// TIA Portal V21 export
ORGANIZATION_BLOCK "Main"   // OB1, LAD, ProgramCycle
TITLE = "Main Program Sweep (Cycle)"
{ S7_Optimized_Access := 'TRUE' }
// stored: SetENOAutomatically false
   VAR_INPUT
      Initial_Call : Bool;   // Initial call of this OB
      Remanence : Bool;   // =True, if remanent data are available
   END_VAR
   VAR_TEMP
      "EQUIPMENT ID" : Variant;
      "EQUIPMENT ID_1" : Variant;
   END_VAR
   VAR_TEMP   // added for the SCL form of the ladder/FBD networks
      _w1 : Bool;
      _w2 : Bool;
      _w3 : Bool;
      _w4 : Bool;
      _w5 : Bool;
      _w6 : Bool;
      _w7 : Bool;
   END_VAR
BEGIN

REGION Network 1: BLOCK CALL
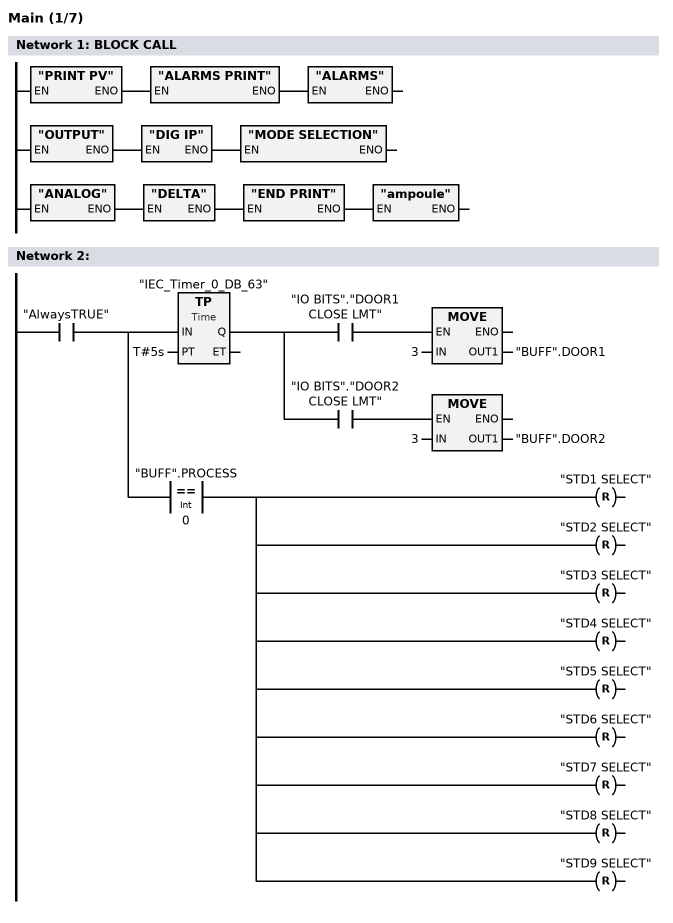
   RUNG wire#powerrail
      "PRINT PV"()
      "ALARMS PRINT"()
      "ALARMS"()
   END_RUNG
   RUNG wire#powerrail
      "OUTPUT"()
      "DIG IP"()
      "MODE SELECTION"()
   END_RUNG
   RUNG wire#powerrail
      "ANALOG"()
      "DELTA"()
      "END PRINT"()
      "ampoule"()
   END_RUNG
   // the same network as SCL:
   "PRINT PV"(ENO => #_w1);
   "ALARMS PRINT"(EN := #_w1, ENO => #_w2);
   IF #_w2 THEN "ALARMS"(); END_IF;
   "OUTPUT"(ENO => #_w3);
   "DIG IP"(EN := #_w3, ENO => #_w4);
   IF #_w4 THEN "MODE SELECTION"(); END_IF;
   "ANALOG"(ENO => #_w5);
   "DELTA"(EN := #_w5, ENO => #_w6);
   "END PRINT"(EN := #_w6, ENO => #_w7);
   IF #_w7 THEN "ampoule"(); END_IF;
END_REGION

REGION Network 2
   RUNG wire#powerrail
      Contact( "AlwaysTRUE" )
      wire#w1
      { S7_Templates := "time_type := Time" } "IEC_Timer_0_DB_63".TP(pt := T#5s, et =>)
      wire#w2
      Contact( "IO BITS"."DOOR1 CLOSE LMT" )
      Move(in := 3, out1 => "BUFF".DOOR1)
   END_RUNG
   RUNG wire#w2
      Contact( "IO BITS"."DOOR2 CLOSE LMT" )
      Move(in := 3, out1 => "BUFF".DOOR2)
   END_RUNG
   RUNG wire#w1
      { S7_Templates := "SrcType := Int" } EQ_Contact(in1 := "BUFF".PROCESS, in2 := 0)
      wire#w3
      R_Coil( "STD1 SELECT" )
   END_RUNG
   RUNG wire#w3
      R_Coil( "STD2 SELECT" )
   END_RUNG
   RUNG wire#w3
      R_Coil( "STD3 SELECT" )
   END_RUNG
   RUNG wire#w3
      R_Coil( "STD4 SELECT" )
   END_RUNG
   RUNG wire#w3
      R_Coil( "STD5 SELECT" )
   END_RUNG
   RUNG wire#w3
      R_Coil( "STD6 SELECT" )
   END_RUNG
   RUNG wire#w3
      R_Coil( "STD7 SELECT" )
   END_RUNG
   RUNG wire#w3
      R_Coil( "STD8 SELECT" )
   END_RUNG
   RUNG wire#w3
      R_Coil( "STD9 SELECT" )
   END_RUNG
   // the same network as SCL:
   "IEC_Timer_0_DB_63".TP(IN := "AlwaysTRUE", PT := T#5s);
   IF "IEC_Timer_0_DB_63".Q AND "IO BITS"."DOOR1 CLOSE LMT" THEN "BUFF".DOOR1 := 3; END_IF;
   IF "IEC_Timer_0_DB_63".Q AND "IO BITS"."DOOR2 CLOSE LMT" THEN "BUFF".DOOR2 := 3; END_IF;
   IF "AlwaysTRUE" AND ("BUFF".PROCESS = 0) THEN
       "STD1 SELECT" := FALSE;
       "STD2 SELECT" := FALSE;
       "STD3 SELECT" := FALSE;
       "STD4 SELECT" := FALSE;
       "STD5 SELECT" := FALSE;
       "STD6 SELECT" := FALSE;
       "STD7 SELECT" := FALSE;
       "STD8 SELECT" := FALSE;
       "STD9 SELECT" := FALSE;
   END_IF;
END_REGION

REGION Network 3: STANDARD1
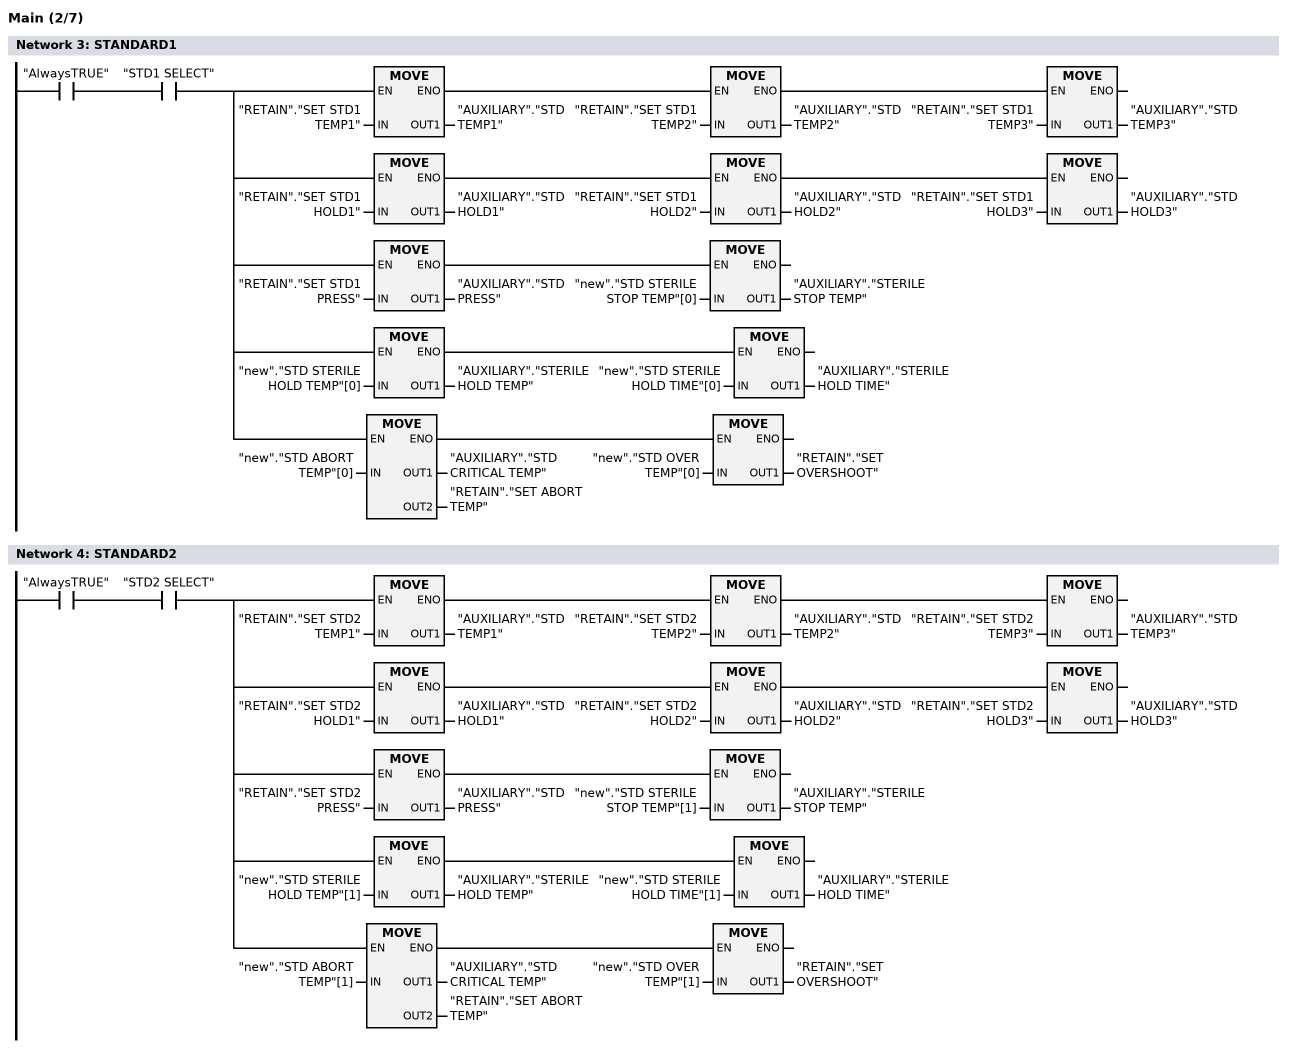
   RUNG wire#powerrail
      Contact( "AlwaysTRUE" )
      Contact( "STD1 SELECT" )
      wire#w1
      Move(in := "RETAIN"."SET STD1 TEMP1", out1 => "AUXILIARY"."STD TEMP1")
      Move(in := "RETAIN"."SET STD1 TEMP2", out1 => "AUXILIARY"."STD TEMP2")
      Move(in := "RETAIN"."SET STD1 TEMP3", out1 => "AUXILIARY"."STD TEMP3")
   END_RUNG
   RUNG wire#w1
      Move(in := "RETAIN"."SET STD1 HOLD1", out1 => "AUXILIARY"."STD HOLD1")
      Move(in := "RETAIN"."SET STD1 HOLD2", out1 => "AUXILIARY"."STD HOLD2")
      Move(in := "RETAIN"."SET STD1 HOLD3", out1 => "AUXILIARY"."STD HOLD3")
   END_RUNG
   RUNG wire#w1
      Move(in := "RETAIN"."SET STD1 PRESS", out1 => "AUXILIARY"."STD PRESS")
      Move(in := "new"."STD STERILE STOP TEMP"[0], out1 => "AUXILIARY"."STERILE STOP TEMP")
   END_RUNG
   RUNG wire#w1
      Move(in := "new"."STD STERILE HOLD TEMP"[0], out1 => "AUXILIARY"."STERILE HOLD TEMP")
      Move(in := "new"."STD STERILE HOLD TIME"[0], out1 => "AUXILIARY"."STERILE HOLD TIME")
   END_RUNG
   RUNG wire#w1
      Move(in := "new"."STD ABORT TEMP"[0], out1 => "AUXILIARY"."STD CRITICAL TEMP", out2 => "RETAIN"."SET ABORT TEMP")
      Move(in := "new"."STD OVER TEMP"[0], out1 => "RETAIN"."SET OVERSHOOT")
   END_RUNG
   // the same network as SCL:
   IF "AlwaysTRUE" AND "STD1 SELECT" THEN
       "AUXILIARY"."STD TEMP1" := "RETAIN"."SET STD1 TEMP1";
       "AUXILIARY"."STD TEMP2" := "RETAIN"."SET STD1 TEMP2";
       "AUXILIARY"."STD TEMP3" := "RETAIN"."SET STD1 TEMP3";
       "AUXILIARY"."STD HOLD1" := "RETAIN"."SET STD1 HOLD1";
       "AUXILIARY"."STD HOLD2" := "RETAIN"."SET STD1 HOLD2";
       "AUXILIARY"."STD HOLD3" := "RETAIN"."SET STD1 HOLD3";
       "AUXILIARY"."STD PRESS" := "RETAIN"."SET STD1 PRESS";
       "AUXILIARY"."STERILE STOP TEMP" := "new"."STD STERILE STOP TEMP"[0];
       "AUXILIARY"."STERILE HOLD TEMP" := "new"."STD STERILE HOLD TEMP"[0];
       "AUXILIARY"."STERILE HOLD TIME" := "new"."STD STERILE HOLD TIME"[0];
       "AUXILIARY"."STD CRITICAL TEMP" := "new"."STD ABORT TEMP"[0];
       "RETAIN"."SET ABORT TEMP" := "new"."STD ABORT TEMP"[0];
       "RETAIN"."SET OVERSHOOT" := "new"."STD OVER TEMP"[0];
   END_IF;
END_REGION

REGION Network 4: STANDARD2
   RUNG wire#powerrail
      Contact( "AlwaysTRUE" )
      Contact( "STD2 SELECT" )
      wire#w1
      Move(in := "RETAIN"."SET STD2 TEMP1", out1 => "AUXILIARY"."STD TEMP1")
      Move(in := "RETAIN"."SET STD2 TEMP2", out1 => "AUXILIARY"."STD TEMP2")
      Move(in := "RETAIN"."SET STD2 TEMP3", out1 => "AUXILIARY"."STD TEMP3")
   END_RUNG
   RUNG wire#w1
      Move(in := "RETAIN"."SET STD2 HOLD1", out1 => "AUXILIARY"."STD HOLD1")
      Move(in := "RETAIN"."SET STD2 HOLD2", out1 => "AUXILIARY"."STD HOLD2")
      Move(in := "RETAIN"."SET STD2 HOLD3", out1 => "AUXILIARY"."STD HOLD3")
   END_RUNG
   RUNG wire#w1
      Move(in := "RETAIN"."SET STD2 PRESS", out1 => "AUXILIARY"."STD PRESS")
      Move(in := "new"."STD STERILE STOP TEMP"[1], out1 => "AUXILIARY"."STERILE STOP TEMP")
   END_RUNG
   RUNG wire#w1
      Move(in := "new"."STD STERILE HOLD TEMP"[1], out1 => "AUXILIARY"."STERILE HOLD TEMP")
      Move(in := "new"."STD STERILE HOLD TIME"[1], out1 => "AUXILIARY"."STERILE HOLD TIME")
   END_RUNG
   RUNG wire#w1
      Move(in := "new"."STD ABORT TEMP"[1], out1 => "AUXILIARY"."STD CRITICAL TEMP", out2 => "RETAIN"."SET ABORT TEMP")
      Move(in := "new"."STD OVER TEMP"[1], out1 => "RETAIN"."SET OVERSHOOT")
   END_RUNG
   // the same network as SCL:
   IF "AlwaysTRUE" AND "STD2 SELECT" THEN
       "AUXILIARY"."STD TEMP1" := "RETAIN"."SET STD2 TEMP1";
       "AUXILIARY"."STD TEMP2" := "RETAIN"."SET STD2 TEMP2";
       "AUXILIARY"."STD TEMP3" := "RETAIN"."SET STD2 TEMP3";
       "AUXILIARY"."STD HOLD1" := "RETAIN"."SET STD2 HOLD1";
       "AUXILIARY"."STD HOLD2" := "RETAIN"."SET STD2 HOLD2";
       "AUXILIARY"."STD HOLD3" := "RETAIN"."SET STD2 HOLD3";
       "AUXILIARY"."STD PRESS" := "RETAIN"."SET STD2 PRESS";
       "AUXILIARY"."STERILE STOP TEMP" := "new"."STD STERILE STOP TEMP"[1];
       "AUXILIARY"."STERILE HOLD TEMP" := "new"."STD STERILE HOLD TEMP"[1];
       "AUXILIARY"."STERILE HOLD TIME" := "new"."STD STERILE HOLD TIME"[1];
       "AUXILIARY"."STD CRITICAL TEMP" := "new"."STD ABORT TEMP"[1];
       "RETAIN"."SET ABORT TEMP" := "new"."STD ABORT TEMP"[1];
       "RETAIN"."SET OVERSHOOT" := "new"."STD OVER TEMP"[1];
   END_IF;
END_REGION

REGION Network 5: STANDARD3
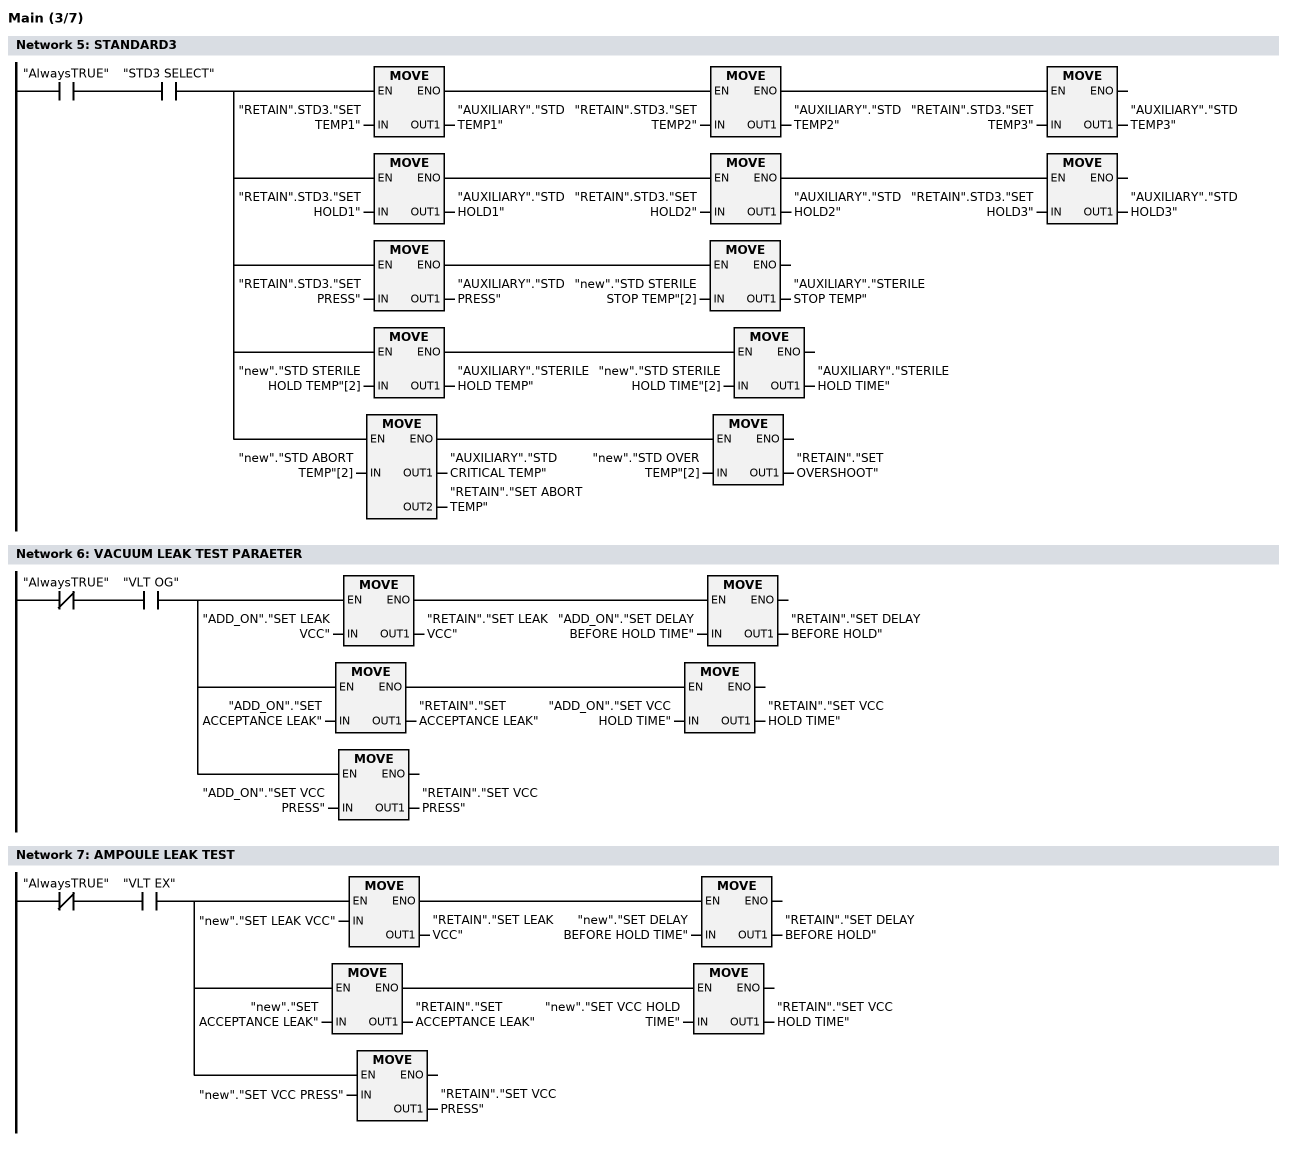
   RUNG wire#powerrail
      Contact( "AlwaysTRUE" )
      Contact( "STD3 SELECT" )
      wire#w1
      Move(in := "RETAIN".STD3."SET TEMP1", out1 => "AUXILIARY"."STD TEMP1")
      Move(in := "RETAIN".STD3."SET TEMP2", out1 => "AUXILIARY"."STD TEMP2")
      Move(in := "RETAIN".STD3."SET TEMP3", out1 => "AUXILIARY"."STD TEMP3")
   END_RUNG
   RUNG wire#w1
      Move(in := "RETAIN".STD3."SET HOLD1", out1 => "AUXILIARY"."STD HOLD1")
      Move(in := "RETAIN".STD3."SET HOLD2", out1 => "AUXILIARY"."STD HOLD2")
      Move(in := "RETAIN".STD3."SET HOLD3", out1 => "AUXILIARY"."STD HOLD3")
   END_RUNG
   RUNG wire#w1
      Move(in := "RETAIN".STD3."SET PRESS", out1 => "AUXILIARY"."STD PRESS")
      Move(in := "new"."STD STERILE STOP TEMP"[2], out1 => "AUXILIARY"."STERILE STOP TEMP")
   END_RUNG
   RUNG wire#w1
      Move(in := "new"."STD STERILE HOLD TEMP"[2], out1 => "AUXILIARY"."STERILE HOLD TEMP")
      Move(in := "new"."STD STERILE HOLD TIME"[2], out1 => "AUXILIARY"."STERILE HOLD TIME")
   END_RUNG
   RUNG wire#w1
      Move(in := "new"."STD ABORT TEMP"[2], out1 => "AUXILIARY"."STD CRITICAL TEMP", out2 => "RETAIN"."SET ABORT TEMP")
      Move(in := "new"."STD OVER TEMP"[2], out1 => "RETAIN"."SET OVERSHOOT")
   END_RUNG
   // the same network as SCL:
   IF "AlwaysTRUE" AND "STD3 SELECT" THEN
       "AUXILIARY"."STD TEMP1" := "RETAIN".STD3."SET TEMP1";
       "AUXILIARY"."STD TEMP2" := "RETAIN".STD3."SET TEMP2";
       "AUXILIARY"."STD TEMP3" := "RETAIN".STD3."SET TEMP3";
       "AUXILIARY"."STD HOLD1" := "RETAIN".STD3."SET HOLD1";
       "AUXILIARY"."STD HOLD2" := "RETAIN".STD3."SET HOLD2";
       "AUXILIARY"."STD HOLD3" := "RETAIN".STD3."SET HOLD3";
       "AUXILIARY"."STD PRESS" := "RETAIN".STD3."SET PRESS";
       "AUXILIARY"."STERILE STOP TEMP" := "new"."STD STERILE STOP TEMP"[2];
       "AUXILIARY"."STERILE HOLD TEMP" := "new"."STD STERILE HOLD TEMP"[2];
       "AUXILIARY"."STERILE HOLD TIME" := "new"."STD STERILE HOLD TIME"[2];
       "AUXILIARY"."STD CRITICAL TEMP" := "new"."STD ABORT TEMP"[2];
       "RETAIN"."SET ABORT TEMP" := "new"."STD ABORT TEMP"[2];
       "RETAIN"."SET OVERSHOOT" := "new"."STD OVER TEMP"[2];
   END_IF;
END_REGION

REGION Network 6: VACUUM LEAK TEST PARAETER
   RUNG wire#powerrail
      I_Contact( "AlwaysTRUE" )
      Contact( "VLT OG" )
      wire#w1
      Move(in := "ADD_ON"."SET LEAK VCC", out1 => "RETAIN"."SET LEAK VCC")
      Move(in := "ADD_ON"."SET DELAY BEFORE HOLD TIME", out1 => "RETAIN"."SET DELAY BEFORE HOLD")
   END_RUNG
   RUNG wire#w1
      Move(in := "ADD_ON"."SET ACCEPTANCE LEAK", out1 => "RETAIN"."SET ACCEPTANCE LEAK")
      Move(in := "ADD_ON"."SET VCC HOLD TIME", out1 => "RETAIN"."SET VCC HOLD TIME")
   END_RUNG
   RUNG wire#w1
      Move(in := "ADD_ON"."SET VCC PRESS", out1 => "RETAIN"."SET VCC PRESS")
   END_RUNG
   // the same network as SCL:
   IF NOT "AlwaysTRUE" AND "VLT OG" THEN
       "RETAIN"."SET LEAK VCC" := "ADD_ON"."SET LEAK VCC";
       "RETAIN"."SET DELAY BEFORE HOLD" := "ADD_ON"."SET DELAY BEFORE HOLD TIME";
       "RETAIN"."SET ACCEPTANCE LEAK" := "ADD_ON"."SET ACCEPTANCE LEAK";
       "RETAIN"."SET VCC HOLD TIME" := "ADD_ON"."SET VCC HOLD TIME";
       "RETAIN"."SET VCC PRESS" := "ADD_ON"."SET VCC PRESS";
   END_IF;
END_REGION

REGION Network 7: AMPOULE LEAK TEST
   RUNG wire#powerrail
      I_Contact( "AlwaysTRUE" )
      Contact( "VLT EX" )
      wire#w1
      Move(in := "new"."SET LEAK VCC", out1 => "RETAIN"."SET LEAK VCC")
      Move(in := "new"."SET DELAY BEFORE HOLD TIME", out1 => "RETAIN"."SET DELAY BEFORE HOLD")
   END_RUNG
   RUNG wire#w1
      Move(in := "new"."SET ACCEPTANCE LEAK", out1 => "RETAIN"."SET ACCEPTANCE LEAK")
      Move(in := "new"."SET VCC HOLD TIME", out1 => "RETAIN"."SET VCC HOLD TIME")
   END_RUNG
   RUNG wire#w1
      Move(in := "new"."SET VCC PRESS", out1 => "RETAIN"."SET VCC PRESS")
   END_RUNG
   // the same network as SCL:
   IF NOT "AlwaysTRUE" AND "VLT EX" THEN
       "RETAIN"."SET LEAK VCC" := "new"."SET LEAK VCC";
       "RETAIN"."SET DELAY BEFORE HOLD" := "new"."SET DELAY BEFORE HOLD TIME";
       "RETAIN"."SET ACCEPTANCE LEAK" := "new"."SET ACCEPTANCE LEAK";
       "RETAIN"."SET VCC HOLD TIME" := "new"."SET VCC HOLD TIME";
       "RETAIN"."SET VCC PRESS" := "new"."SET VCC PRESS";
   END_IF;
END_REGION

REGION Network 8: MONTH_L
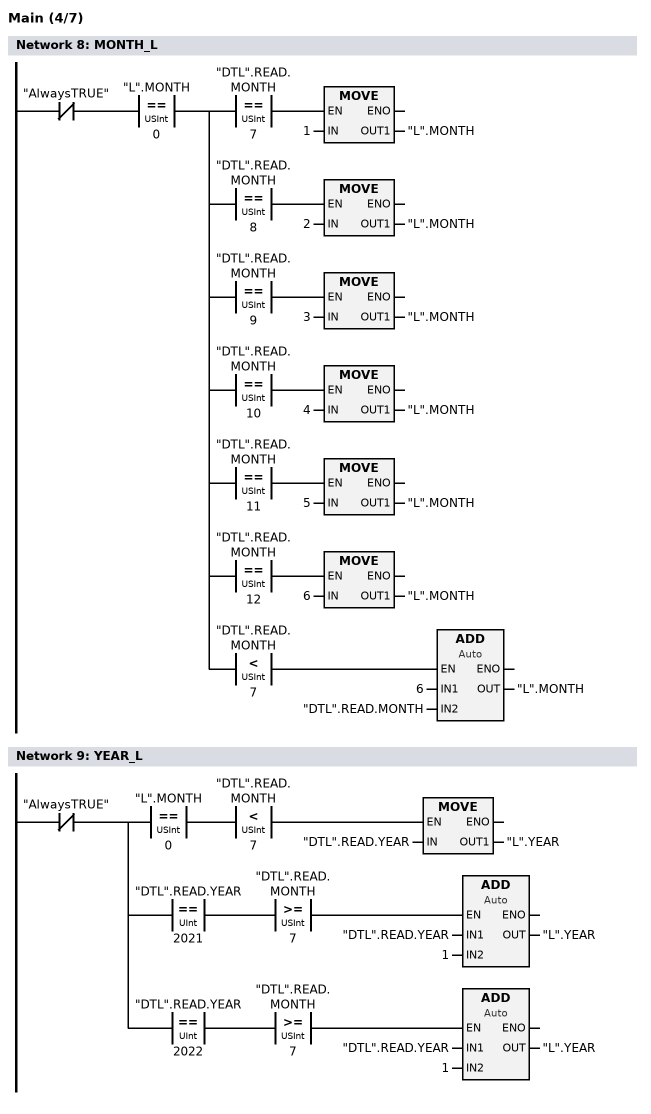
   RUNG wire#powerrail
      I_Contact( "AlwaysTRUE" )
      { S7_Templates := "SrcType := USInt" } EQ_Contact(in1 := "L".MONTH, in2 := 0)
      wire#w1
      { S7_Templates := "SrcType := USInt" } EQ_Contact(in1 := "DTL".READ.MONTH, in2 := 7)
      Move(in := 1, out1 => "L".MONTH)
   END_RUNG
   RUNG wire#w1
      { S7_Templates := "SrcType := USInt" } EQ_Contact(in1 := "DTL".READ.MONTH, in2 := 8)
      Move(in := 2, out1 => "L".MONTH)
   END_RUNG
   RUNG wire#w1
      { S7_Templates := "SrcType := USInt" } EQ_Contact(in1 := "DTL".READ.MONTH, in2 := 9)
      Move(in := 3, out1 => "L".MONTH)
   END_RUNG
   RUNG wire#w1
      { S7_Templates := "SrcType := USInt" } EQ_Contact(in1 := "DTL".READ.MONTH, in2 := 10)
      Move(in := 4, out1 => "L".MONTH)
   END_RUNG
   RUNG wire#w1
      { S7_Templates := "SrcType := USInt" } EQ_Contact(in1 := "DTL".READ.MONTH, in2 := 11)
      Move(in := 5, out1 => "L".MONTH)
   END_RUNG
   RUNG wire#w1
      { S7_Templates := "SrcType := USInt" } EQ_Contact(in1 := "DTL".READ.MONTH, in2 := 12)
      Move(in := 6, out1 => "L".MONTH)
   END_RUNG
   RUNG wire#w1
      { S7_Templates := "SrcType := USInt" } LT_Contact(in1 := "DTL".READ.MONTH, in2 := 7)
      Add(in1 := 6, in2 := "DTL".READ.MONTH, out => "L".MONTH)
   END_RUNG
   // the same network as SCL:
   #_w1 := NOT "AlwaysTRUE" AND ("L".MONTH = 0);
   IF #_w1 AND ("DTL".READ.MONTH = 7) THEN "L".MONTH := 1; END_IF;
   IF #_w1 AND ("DTL".READ.MONTH = 8) THEN "L".MONTH := 2; END_IF;
   IF #_w1 AND ("DTL".READ.MONTH = 9) THEN "L".MONTH := 3; END_IF;
   IF #_w1 AND ("DTL".READ.MONTH = 10) THEN "L".MONTH := 4; END_IF;
   IF #_w1 AND ("DTL".READ.MONTH = 11) THEN "L".MONTH := 5; END_IF;
   IF #_w1 AND ("DTL".READ.MONTH = 12) THEN "L".MONTH := 6; END_IF;
   IF #_w1 AND ("DTL".READ.MONTH < 7) THEN "L".MONTH := 6 + "DTL".READ.MONTH; END_IF;
END_REGION

REGION Network 9: YEAR_L
   RUNG wire#powerrail
      I_Contact( "AlwaysTRUE" )
      wire#w1
      { S7_Templates := "SrcType := USInt" } EQ_Contact(in1 := "L".MONTH, in2 := 0)
      { S7_Templates := "SrcType := USInt" } LT_Contact(in1 := "DTL".READ.MONTH, in2 := 7)
      Move(in := "DTL".READ.YEAR, out1 => "L".YEAR)
   END_RUNG
   RUNG wire#w1
      { S7_Templates := "SrcType := UInt" } EQ_Contact(in1 := "DTL".READ.YEAR, in2 := 2021)
      { S7_Templates := "SrcType := USInt" } GE_Contact(in1 := "DTL".READ.MONTH, in2 := 7)
      Add(in1 := "DTL".READ.YEAR, in2 := 1, out => "L".YEAR)
   END_RUNG
   RUNG wire#w1
      { S7_Templates := "SrcType := UInt" } EQ_Contact(in1 := "DTL".READ.YEAR, in2 := 2022)
      { S7_Templates := "SrcType := USInt" } GE_Contact(in1 := "DTL".READ.MONTH, in2 := 7)
      Add(in1 := "DTL".READ.YEAR, in2 := 1, out => "L".YEAR)
   END_RUNG
   // the same network as SCL:
   IF NOT "AlwaysTRUE" AND ("L".MONTH = 0) AND ("DTL".READ.MONTH < 7) THEN
       "L".YEAR := "DTL".READ.YEAR;
   END_IF;
   IF NOT "AlwaysTRUE" AND ("DTL".READ.YEAR = 2021) AND ("DTL".READ.MONTH >= 7) THEN
       "L".YEAR := "DTL".READ.YEAR + 1;
   END_IF;
   IF NOT "AlwaysTRUE" AND ("DTL".READ.YEAR = 2022) AND ("DTL".READ.MONTH >= 7) THEN
       "L".YEAR := "DTL".READ.YEAR + 1;
   END_IF;
END_REGION

REGION Network 10: IMP
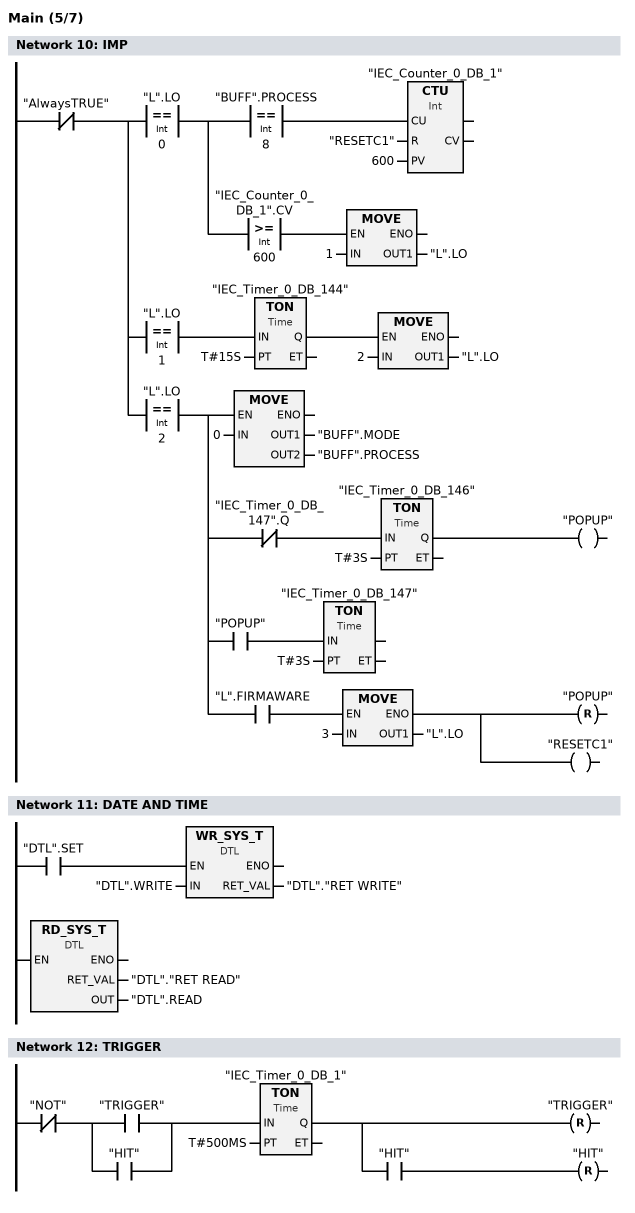
   RUNG wire#powerrail
      I_Contact( "AlwaysTRUE" )
      wire#w1
      { S7_Templates := "SrcType := Int" } EQ_Contact(in1 := "L".LO, in2 := 0)
      wire#w2
      { S7_Templates := "SrcType := Int" } EQ_Contact(in1 := "BUFF".PROCESS, in2 := 8)
      { S7_Templates := "value_type := Int" } "IEC_Counter_0_DB_1".CTU(r := "RESETC1", pv := 600, cv =>)
   END_RUNG
   RUNG wire#w2
      { S7_Templates := "SrcType := Int" } GE_Contact(in1 := "IEC_Counter_0_DB_1".CV, in2 := 600)
      Move(in := 1, out1 => "L".LO)
   END_RUNG
   RUNG wire#w1
      { S7_Templates := "SrcType := Int" } EQ_Contact(in1 := "L".LO, in2 := 1)
      { S7_Templates := "time_type := Time" } "IEC_Timer_0_DB_144".TON(pt := T#15S, et =>)
      Move(in := 2, out1 => "L".LO)
   END_RUNG
   RUNG wire#w1
      { S7_Templates := "SrcType := Int" } EQ_Contact(in1 := "L".LO, in2 := 2)
      wire#w3
      Move(in := 0, out1 => "BUFF".MODE, out2 => "BUFF".PROCESS)
   END_RUNG
   RUNG wire#w3
      I_Contact( "IEC_Timer_0_DB_147".Q )
      { S7_Templates := "time_type := Time" } "IEC_Timer_0_DB_146".TON(pt := T#3S, et =>)
      Coil( "POPUP" )
   END_RUNG
   RUNG wire#w3
      Contact( "POPUP" )
      { S7_Templates := "time_type := Time" } "IEC_Timer_0_DB_147".TON(pt := T#3S, et =>)
   END_RUNG
   RUNG wire#w3
      Contact( "L".FIRMAWARE )
      Move(in := 3, out1 => "L".LO)
      wire#w4
      R_Coil( "POPUP" )
   END_RUNG
   RUNG wire#w4
      Coil( "RESETC1" )
   END_RUNG
   // the same network as SCL:
   #_w1 := NOT "AlwaysTRUE" AND ("L".LO = 0);
   "IEC_Counter_0_DB_1".CTU(CU := #_w1 AND ("BUFF".PROCESS = 8), R := "RESETC1", PV := 600);
   IF #_w1 AND ("IEC_Counter_0_DB_1".CV >= 600) THEN "L".LO := 1; END_IF;
   "IEC_Timer_0_DB_144".TON(IN := NOT "AlwaysTRUE" AND ("L".LO = 1), PT := T#15S);
   IF "IEC_Timer_0_DB_144".Q THEN "L".LO := 2; END_IF;
   #_w2 := NOT "AlwaysTRUE" AND ("L".LO = 2);
   IF #_w2 THEN
       "BUFF".MODE := 0;
       "BUFF".PROCESS := 0;
   END_IF;
   "IEC_Timer_0_DB_146".TON(IN := #_w2 AND NOT "IEC_Timer_0_DB_147".Q, PT := T#3S);
   "POPUP" := "IEC_Timer_0_DB_146".Q;
   "IEC_Timer_0_DB_147".TON(IN := #_w2 AND "POPUP", PT := T#3S);
   #_w3 := #_w2 AND "L".FIRMAWARE;
   IF #_w3 THEN
       "L".LO := 3;
       "POPUP" := FALSE;
   END_IF;
   "RESETC1" := #_w3;
END_REGION

REGION Network 11: DATE AND TIME
   RUNG wire#powerrail
      Contact( "DTL".SET )
      { S7_Templates := "date_type := DTL" } WR_SYS_T(IN := "DTL".WRITE, RET_VAL => "DTL"."RET WRITE")
   END_RUNG
   RUNG wire#powerrail
      { S7_Templates := "date_type := DTL" } RD_SYS_T(RET_VAL => "DTL"."RET READ", OUT => "DTL".READ)
   END_RUNG
   // the same network as SCL:
   IF "DTL".SET THEN "DTL"."RET WRITE" := WR_SYS_T(IN := "DTL".WRITE); END_IF;
   "DTL"."RET READ" := RD_SYS_T(OUT => "DTL".READ);
END_REGION

REGION Network 12: TRIGGER
   RUNG wire#powerrail
      I_Contact( "NOT" )
      wire#w1
      Contact( "TRIGGER" )
      wire#w2
      { S7_Templates := "time_type := Time" } "IEC_Timer_0_DB_1".TON(pt := T#500MS, et =>)
      wire#w3
      R_Coil( "TRIGGER" )
   END_RUNG
   RUNG wire#w1
      Contact( "HIT" )
   END_RUNG wire#w2
   RUNG wire#w3
      Contact( "HIT" )
      R_Coil( "HIT" )
   END_RUNG
   // the same network as SCL:
   "IEC_Timer_0_DB_1".TON(IN := NOT "NOT" AND ("TRIGGER" OR "HIT"), PT := T#500MS);
   IF "IEC_Timer_0_DB_1".Q THEN "TRIGGER" := FALSE; END_IF;
   IF "IEC_Timer_0_DB_1".Q AND "HIT" THEN "HIT" := FALSE; END_IF;
END_REGION

REGION Network 13: CYCLE COUNT
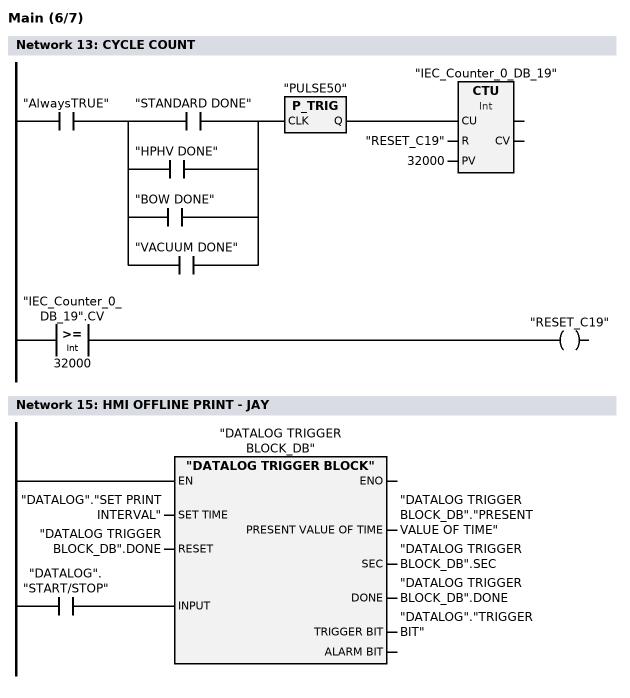
   RUNG wire#powerrail
      Contact( "AlwaysTRUE" )
      wire#w1
      Contact( "STANDARD DONE" )
      wire#w2
      P_Trig( "PULSE50" )
      { S7_Templates := "value_type := Int" } "IEC_Counter_0_DB_19".CTU(r := "RESET_C19", pv := 32000, cv =>)
   END_RUNG
   RUNG wire#w1
      Contact( "HPHV DONE" )
   END_RUNG wire#w2
   RUNG wire#w1
      Contact( "BOW DONE" )
   END_RUNG wire#w2
   RUNG wire#w1
      Contact( "VACUUM DONE" )
   END_RUNG wire#w2
   RUNG wire#powerrail
      { S7_Templates := "SrcType := Int" } GE_Contact(in1 := "IEC_Counter_0_DB_19".CV, in2 := 32000)
      Coil( "RESET_C19" )
   END_RUNG
   // the same network as SCL:
   #_w1 := "AlwaysTRUE" AND ("STANDARD DONE" OR "HPHV DONE" OR "BOW DONE" OR "VACUUM DONE");
   #_w2 := #_w1 AND NOT "PULSE50";   // rising edge
   "PULSE50" := #_w1;
   "IEC_Counter_0_DB_19".CTU(CU := #_w2, R := "RESET_C19", PV := 32000);
   "RESET_C19" := "IEC_Counter_0_DB_19".CV >= 32000;
END_REGION

REGION Network 15: HMI OFFLINE PRINT - JAY
   RUNG wire#powerrail
      "DATALOG TRIGGER BLOCK_DB"(INPUT := wire#w1, "SET TIME" := "DATALOG"."SET PRINT INTERVAL", RESET := "DATALOG TRIGGER BLOCK_DB".DONE, "PRESENT VALUE OF TIME" => "DATALOG TRIGGER BLOCK_DB"."PRESENT VALUE OF TIME", SEC => "DATALOG TRIGGER BLOCK_DB".SEC, DONE => "DATALOG TRIGGER BLOCK_DB".DONE, "TRIGGER BIT" => "DATALOG"."TRIGGER BIT", "ALARM BIT" =>)
   END_RUNG
   RUNG wire#powerrail
      Contact( "DATALOG"."START/STOP" )
   END_RUNG wire#w1
   // the same network as SCL:
   "DATALOG TRIGGER BLOCK_DB"("SET TIME" := "DATALOG"."SET PRINT INTERVAL",   // "DATALOG TRIGGER BLOCK"
                           RESET := "DATALOG TRIGGER BLOCK_DB".DONE,
                           INPUT := "DATALOG"."START/STOP",
                           "PRESENT VALUE OF TIME" => "DATALOG TRIGGER BLOCK_DB"."PRESENT VALUE OF TIME",
                           SEC => "DATALOG TRIGGER BLOCK_DB".SEC,
                           DONE => "DATALOG TRIGGER BLOCK_DB".DONE,
                           "TRIGGER BIT" => "DATALOG"."TRIGGER BIT");
END_REGION

REGION Network 16: BATCH START STOP INTERLOCK
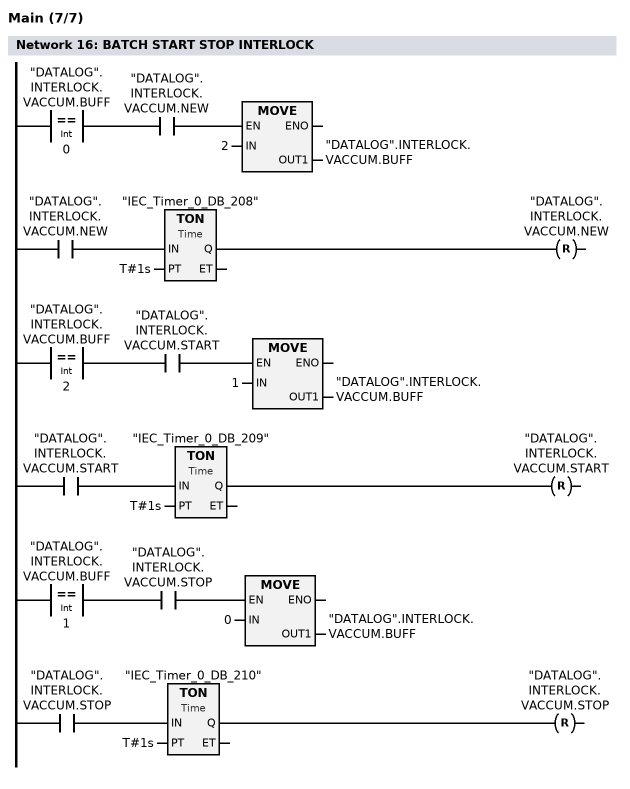
   RUNG wire#powerrail
      { S7_Templates := "SrcType := Int" } EQ_Contact(in1 := "DATALOG".INTERLOCK.VACCUM.BUFF, in2 := 0)
      Contact( "DATALOG".INTERLOCK.VACCUM.NEW )
      Move(in := 2, out1 => "DATALOG".INTERLOCK.VACCUM.BUFF)
   END_RUNG
   RUNG wire#powerrail
      Contact( "DATALOG".INTERLOCK.VACCUM.NEW )
      { S7_Templates := "time_type := Time" } "IEC_Timer_0_DB_208".TON(pt := T#1s, et =>)
      R_Coil( "DATALOG".INTERLOCK.VACCUM.NEW )
   END_RUNG
   RUNG wire#powerrail
      { S7_Templates := "SrcType := Int" } EQ_Contact(in1 := "DATALOG".INTERLOCK.VACCUM.BUFF, in2 := 2)
      Contact( "DATALOG".INTERLOCK.VACCUM.START )
      Move(in := 1, out1 => "DATALOG".INTERLOCK.VACCUM.BUFF)
   END_RUNG
   RUNG wire#powerrail
      Contact( "DATALOG".INTERLOCK.VACCUM.START )
      { S7_Templates := "time_type := Time" } "IEC_Timer_0_DB_209".TON(pt := T#1s, et =>)
      R_Coil( "DATALOG".INTERLOCK.VACCUM.START )
   END_RUNG
   RUNG wire#powerrail
      { S7_Templates := "SrcType := Int" } EQ_Contact(in1 := "DATALOG".INTERLOCK.VACCUM.BUFF, in2 := 1)
      Contact( "DATALOG".INTERLOCK.VACCUM.STOP )
      Move(in := 0, out1 => "DATALOG".INTERLOCK.VACCUM.BUFF)
   END_RUNG
   RUNG wire#powerrail
      Contact( "DATALOG".INTERLOCK.VACCUM.STOP )
      { S7_Templates := "time_type := Time" } "IEC_Timer_0_DB_210".TON(pt := T#1s, et =>)
      R_Coil( "DATALOG".INTERLOCK.VACCUM.STOP )
   END_RUNG
   // the same network as SCL:
   IF ("DATALOG".INTERLOCK.VACCUM.BUFF = 0) AND "DATALOG".INTERLOCK.VACCUM.NEW THEN
       "DATALOG".INTERLOCK.VACCUM.BUFF := 2;
   END_IF;
   "IEC_Timer_0_DB_208".TON(IN := "DATALOG".INTERLOCK.VACCUM.NEW, PT := T#1s);
   IF "IEC_Timer_0_DB_208".Q THEN "DATALOG".INTERLOCK.VACCUM.NEW := FALSE; END_IF;
   IF ("DATALOG".INTERLOCK.VACCUM.BUFF = 2) AND "DATALOG".INTERLOCK.VACCUM.START THEN
       "DATALOG".INTERLOCK.VACCUM.BUFF := 1;
   END_IF;
   "IEC_Timer_0_DB_209".TON(IN := "DATALOG".INTERLOCK.VACCUM.START, PT := T#1s);
   IF "IEC_Timer_0_DB_209".Q THEN "DATALOG".INTERLOCK.VACCUM.START := FALSE; END_IF;
   IF ("DATALOG".INTERLOCK.VACCUM.BUFF = 1) AND "DATALOG".INTERLOCK.VACCUM.STOP THEN
       "DATALOG".INTERLOCK.VACCUM.BUFF := 0;
   END_IF;
   "IEC_Timer_0_DB_210".TON(IN := "DATALOG".INTERLOCK.VACCUM.STOP, PT := T#1s);
   IF "IEC_Timer_0_DB_210".Q THEN "DATALOG".INTERLOCK.VACCUM.STOP := FALSE; END_IF;
END_REGION
END_ORGANIZATION_BLOCK
